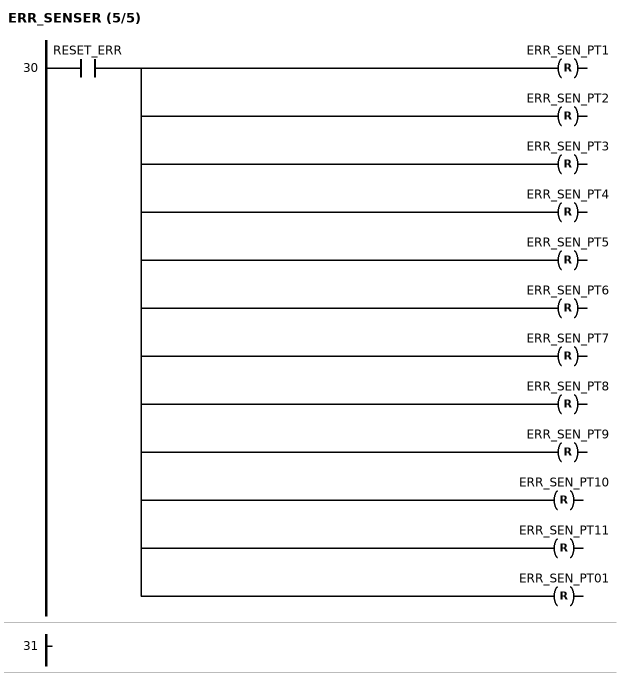
// NETWORK 30
ERR_SEN_PT1 R= RESET_ERR;
ERR_SEN_PT2 R= RESET_ERR;
ERR_SEN_PT3 R= RESET_ERR;
ERR_SEN_PT4 R= RESET_ERR;
ERR_SEN_PT5 R= RESET_ERR;
ERR_SEN_PT6 R= RESET_ERR;
ERR_SEN_PT7 R= RESET_ERR;
ERR_SEN_PT8 R= RESET_ERR;
ERR_SEN_PT9 R= RESET_ERR;
ERR_SEN_PT10 R= RESET_ERR;
ERR_SEN_PT11 R= RESET_ERR;
ERR_SEN_PT01 R= RESET_ERR;

// NETWORK 31

END_PROGRAM

// MyController/Application/SECURITY_BOILER
PROGRAM SECURITY_BOILER
VAR
END_VAR
VAR // added by the converter: edge detectors and wires of the graphical bodies
    _rt1, _rt2, _rt3, _rt4, _rt5 : R_TRIG;
END_VAR

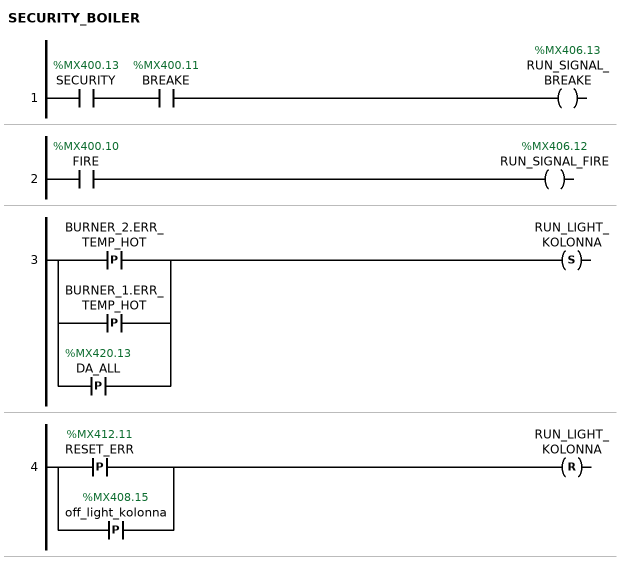
// NETWORK 1
//   SECURITY: AT %MX400.13
//   BREAKE: AT %MX400.11
//   RUN_SIGNAL_BREAKE: AT %MX406.13
RUN_SIGNAL_BREAKE := SECURITY AND BREAKE;

// NETWORK 2
//   FIRE: AT %MX400.10
//   RUN_SIGNAL_FIRE: AT %MX406.12
RUN_SIGNAL_FIRE := FIRE;

// NETWORK 3
//   DA_ALL: AT %MX420.13
_rt1(CLK := BURNER_2.ERR_TEMP_HOT);
_rt2(CLK := BURNER_1.ERR_TEMP_HOT);
_rt3(CLK := DA_ALL);
RUN_LIGHT_KOLONNA S= _rt1.Q OR _rt2.Q OR _rt3.Q;

// NETWORK 4
//   RESET_ERR: AT %MX412.11
//   off_light_kolonna: AT %MX408.15
_rt4(CLK := RESET_ERR);
_rt5(CLK := off_light_kolonna);
RUN_LIGHT_KOLONNA R= _rt4.Q OR _rt5.Q;

END_PROGRAM

// MyController/Application/VALVE_FEEDER_PUMP_FEEDERS_M3_M4
PROGRAM VALVE_FEEDER_PUMP_FEEDERS_M3_M4
VAR
	FEEDER_M3_CYCLE: BOOL;
	FEEDER_M4_CYCLE: BOOL;
	SMALL_PRESS: BOOL;
	run_feeder_to_open: BOOL;
END_VAR
VAR // added by the converter: edge detectors and wires of the graphical bodies
    _rt1, _rt2 : R_TRIG;
    _w1, _w2 : BOOL;
END_VAR

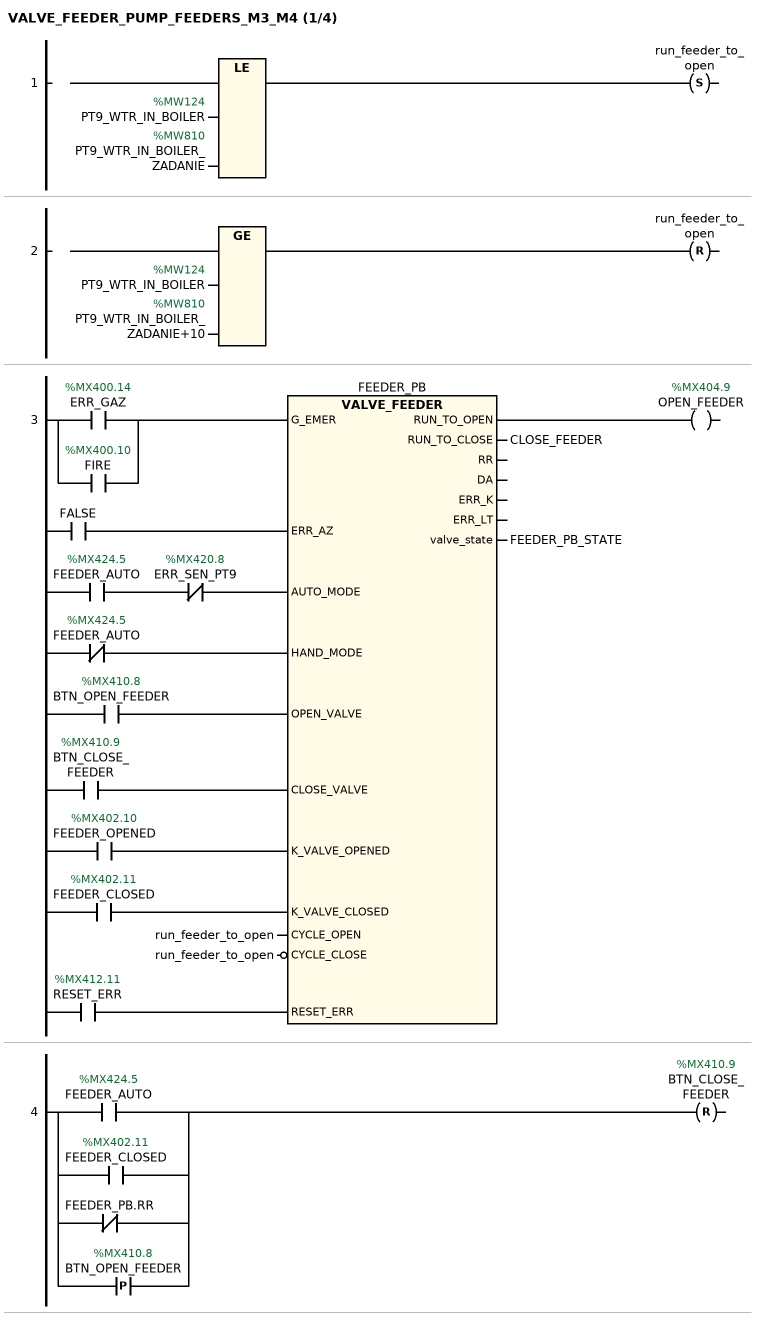
// NETWORK 1
//   PT9_WTR_IN_BOILER: AT %MW124
//   PT9_WTR_IN_BOILER_ZADANIE: AT %MW810
run_feeder_to_open S= PT9_WTR_IN_BOILER <= PT9_WTR_IN_BOILER_ZADANIE;

// NETWORK 2
//   PT9_WTR_IN_BOILER: AT %MW124
//   PT9_WTR_IN_BOILER_ZADANIE+10: AT %MW810
run_feeder_to_open R= PT9_WTR_IN_BOILER >= (PT9_WTR_IN_BOILER_ZADANIE+10);

// NETWORK 3
//   ERR_GAZ: AT %MX400.14
//   FIRE: AT %MX400.10
//   FEEDER_AUTO: AT %MX424.5
//   ERR_SEN_PT9: AT %MX420.8
//   BTN_OPEN_FEEDER: AT %MX410.8
//   BTN_CLOSE_FEEDER: AT %MX410.9
//   FEEDER_OPENED: AT %MX402.10
//   FEEDER_CLOSED: AT %MX402.11
//   RESET_ERR: AT %MX412.11
//   CLOSE_FEEDER: AT %MX404.10
//   FEEDER_PB_STATE: AT %MW406
//   OPEN_FEEDER: AT %MX404.9
FEEDER_PB(
    G_EMER := ERR_GAZ OR FIRE,
    ERR_AZ := FALSE,
    AUTO_MODE := FEEDER_AUTO AND NOT ERR_SEN_PT9,
    HAND_MODE := NOT FEEDER_AUTO,
    OPEN_VALVE := BTN_OPEN_FEEDER,
    CLOSE_VALVE := BTN_CLOSE_FEEDER,
    K_VALVE_OPENED := FEEDER_OPENED,
    K_VALVE_CLOSED := FEEDER_CLOSED,
    CYCLE_OPEN := run_feeder_to_open,
    CYCLE_CLOSE := NOT run_feeder_to_open,
    RESET_ERR := RESET_ERR,
    RUN_TO_CLOSE => CLOSE_FEEDER,
    valve_state => FEEDER_PB_STATE); // VALVE_FEEDER
OPEN_FEEDER := FEEDER_PB.RUN_TO_OPEN;

// NETWORK 4
//   FEEDER_AUTO: AT %MX424.5
//   FEEDER_CLOSED: AT %MX402.11
//   BTN_OPEN_FEEDER: AT %MX410.8
//   BTN_CLOSE_FEEDER: AT %MX410.9
_rt1(CLK := BTN_OPEN_FEEDER);
BTN_CLOSE_FEEDER R= FEEDER_AUTO OR FEEDER_CLOSED OR NOT FEEDER_PB.RR OR _rt1.Q;

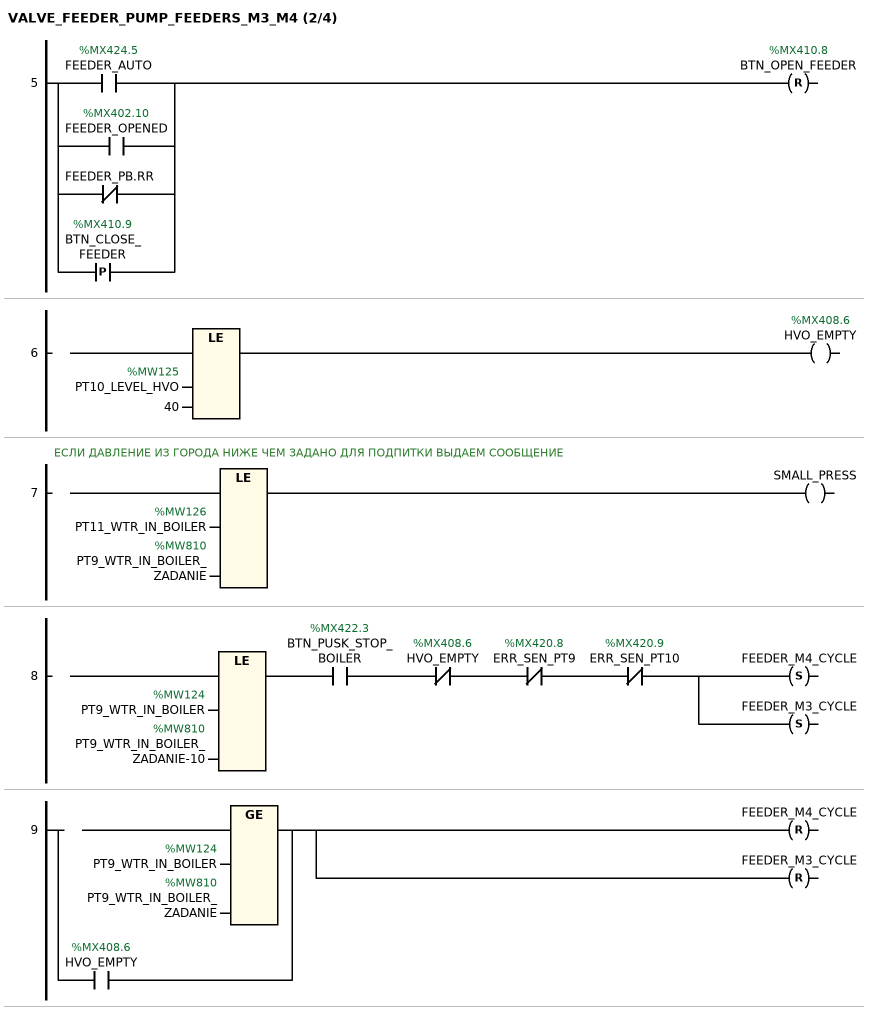
// NETWORK 5
//   FEEDER_AUTO: AT %MX424.5
//   FEEDER_OPENED: AT %MX402.10
//   BTN_CLOSE_FEEDER: AT %MX410.9
//   BTN_OPEN_FEEDER: AT %MX410.8
_rt2(CLK := BTN_CLOSE_FEEDER);
BTN_OPEN_FEEDER R= FEEDER_AUTO OR FEEDER_OPENED OR NOT FEEDER_PB.RR OR _rt2.Q;

// NETWORK 6
//   PT10_LEVEL_HVO: AT %MW125
//   HVO_EMPTY: AT %MX408.6
HVO_EMPTY := PT10_LEVEL_HVO <= 40;

// NETWORK 7
// ЕСЛИ ДАВЛЕНИЕ ИЗ ГОРОДА НИЖЕ ЧЕМ ЗАДАНО ДЛЯ ПОДПИТКИ ВЫДАЕМ СООБЩЕНИЕ
//   PT11_WTR_IN_BOILER: AT %MW126
//   PT9_WTR_IN_BOILER_ZADANIE: AT %MW810
SMALL_PRESS := PT11_WTR_IN_BOILER <= PT9_WTR_IN_BOILER_ZADANIE;

// NETWORK 8
//   PT9_WTR_IN_BOILER: AT %MW124
//   PT9_WTR_IN_BOILER_ZADANIE-10: AT %MW810
//   BTN_PUSK_STOP_BOILER: AT %MX422.3
//   HVO_EMPTY: AT %MX408.6
//   ERR_SEN_PT9: AT %MX420.8
//   ERR_SEN_PT10: AT %MX420.9
_w1 := PT9_WTR_IN_BOILER <= (PT9_WTR_IN_BOILER_ZADANIE-10) AND BTN_PUSK_STOP_BOILER AND NOT HVO_EMPTY AND NOT ERR_SEN_PT9 AND NOT ERR_SEN_PT10;
FEEDER_M4_CYCLE S= _w1;
FEEDER_M3_CYCLE S= _w1;

// NETWORK 9
//   PT9_WTR_IN_BOILER: AT %MW124
//   PT9_WTR_IN_BOILER_ZADANIE: AT %MW810
//   HVO_EMPTY: AT %MX408.6
_w2 := PT9_WTR_IN_BOILER >= PT9_WTR_IN_BOILER_ZADANIE OR HVO_EMPTY;
FEEDER_M4_CYCLE R= _w2;
FEEDER_M3_CYCLE R= _w2;

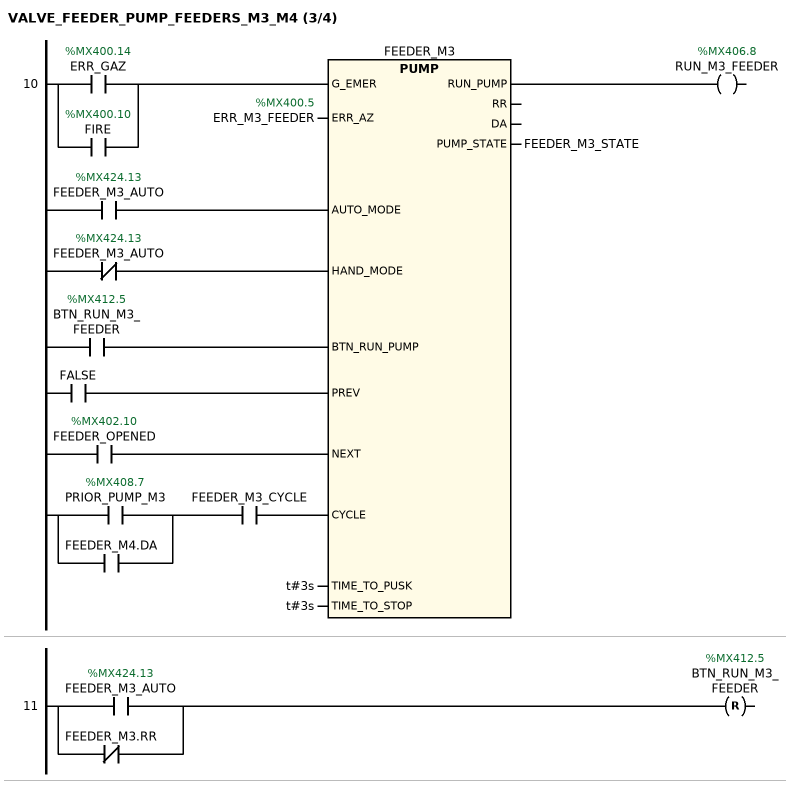
// NETWORK 10
//   ERR_GAZ: AT %MX400.14
//   FIRE: AT %MX400.10
//   ERR_M3_FEEDER: AT %MX400.5
//   FEEDER_M3_AUTO: AT %MX424.13
//   BTN_RUN_M3_FEEDER: AT %MX412.5
//   FEEDER_OPENED: AT %MX402.10
//   PRIOR_PUMP_M3: AT %MX408.7
//   FEEDER_M3_STATE: AT %MW411
//   RUN_M3_FEEDER: AT %MX406.8
FEEDER_M3(
    G_EMER := ERR_GAZ OR FIRE,
    ERR_AZ := ERR_M3_FEEDER,
    AUTO_MODE := FEEDER_M3_AUTO,
    HAND_MODE := NOT FEEDER_M3_AUTO,
    BTN_RUN_PUMP := BTN_RUN_M3_FEEDER,
    PREV := FALSE,
    NEXT := FEEDER_OPENED,
    CYCLE := (PRIOR_PUMP_M3 OR FEEDER_M4.DA) AND FEEDER_M3_CYCLE,
    TIME_TO_PUSK := t#3s,
    TIME_TO_STOP := t#3s,
    PUMP_STATE => FEEDER_M3_STATE); // PUMP
RUN_M3_FEEDER := FEEDER_M3.RUN_PUMP;

// NETWORK 11
//   FEEDER_M3_AUTO: AT %MX424.13
//   BTN_RUN_M3_FEEDER: AT %MX412.5
BTN_RUN_M3_FEEDER R= FEEDER_M3_AUTO OR NOT FEEDER_M3.RR;

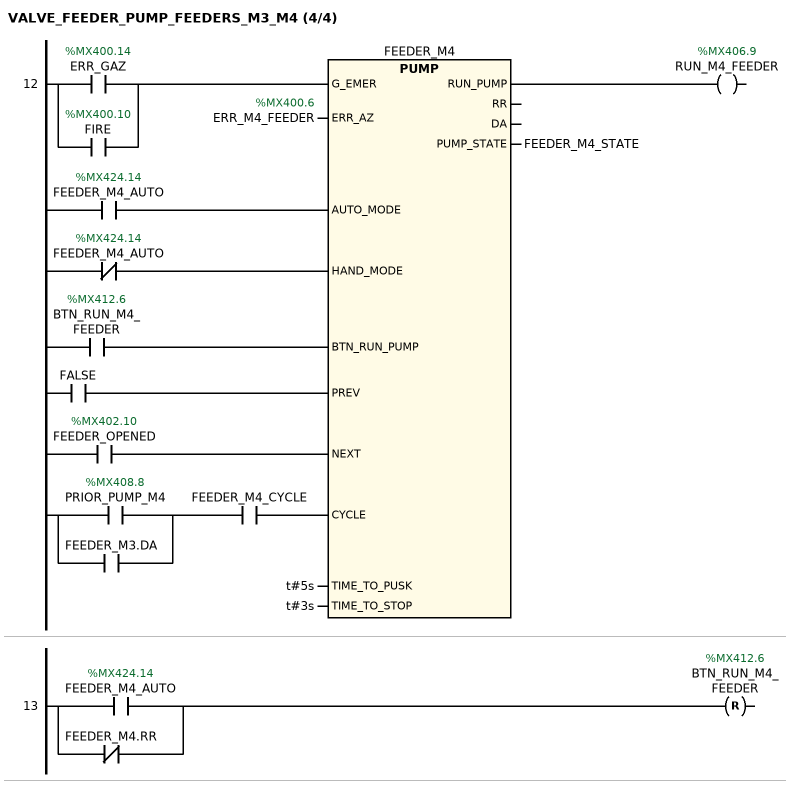
// NETWORK 12
//   ERR_GAZ: AT %MX400.14
//   FIRE: AT %MX400.10
//   ERR_M4_FEEDER: AT %MX400.6
//   FEEDER_M4_AUTO: AT %MX424.14
//   BTN_RUN_M4_FEEDER: AT %MX412.6
//   FEEDER_OPENED: AT %MX402.10
//   PRIOR_PUMP_M4: AT %MX408.8
//   FEEDER_M4_STATE: AT %MW412
//   RUN_M4_FEEDER: AT %MX406.9
FEEDER_M4(
    G_EMER := ERR_GAZ OR FIRE,
    ERR_AZ := ERR_M4_FEEDER,
    AUTO_MODE := FEEDER_M4_AUTO,
    HAND_MODE := NOT FEEDER_M4_AUTO,
    BTN_RUN_PUMP := BTN_RUN_M4_FEEDER,
    PREV := FALSE,
    NEXT := FEEDER_OPENED,
    CYCLE := (PRIOR_PUMP_M4 OR FEEDER_M3.DA) AND FEEDER_M4_CYCLE,
    TIME_TO_PUSK := t#5s,
    TIME_TO_STOP := t#3s,
    PUMP_STATE => FEEDER_M4_STATE); // PUMP
RUN_M4_FEEDER := FEEDER_M4.RUN_PUMP;

// NETWORK 13
//   FEEDER_M4_AUTO: AT %MX424.14
//   BTN_RUN_M4_FEEDER: AT %MX412.6
BTN_RUN_M4_FEEDER R= FEEDER_M4_AUTO OR NOT FEEDER_M4.RR;

END_PROGRAM

// MyController/Application/FB/VALVE_FEEDER
FUNCTION_BLOCK VALVE_FEEDER
VAR_INPUT
	G_EMER: BOOL;
	ERR_AZ: BOOL;
	AUTO_MODE: BOOL;
	HAND_MODE: BOOL;
	OPEN_VALVE: BOOL;
	CLOSE_VALVE: BOOL;
	K_VALVE_OPENED: BOOL;
	K_VALVE_CLOSED: BOOL;
	CYCLE_OPEN: BOOL;
	CYCLE_CLOSE: BOOL;
	RESET_ERR: BOOL;	
END_VAR
VAR_OUTPUT
	RUN_TO_OPEN: BOOL;
	RUN_TO_CLOSE: BOOL;
	RR: BOOL;
	DA: BOOL;
	ERR_K: BOOL;
	ERR_LT: BOOL;
	valve_state: BYTE;
END_VAR
VAR
	TM_LT_VALVE: TON;
	tm_err_k: TOF;
END_VAR
VAR // added by the converter: edge detectors and wires of the graphical bodies
    _w1 : BOOL;
END_VAR

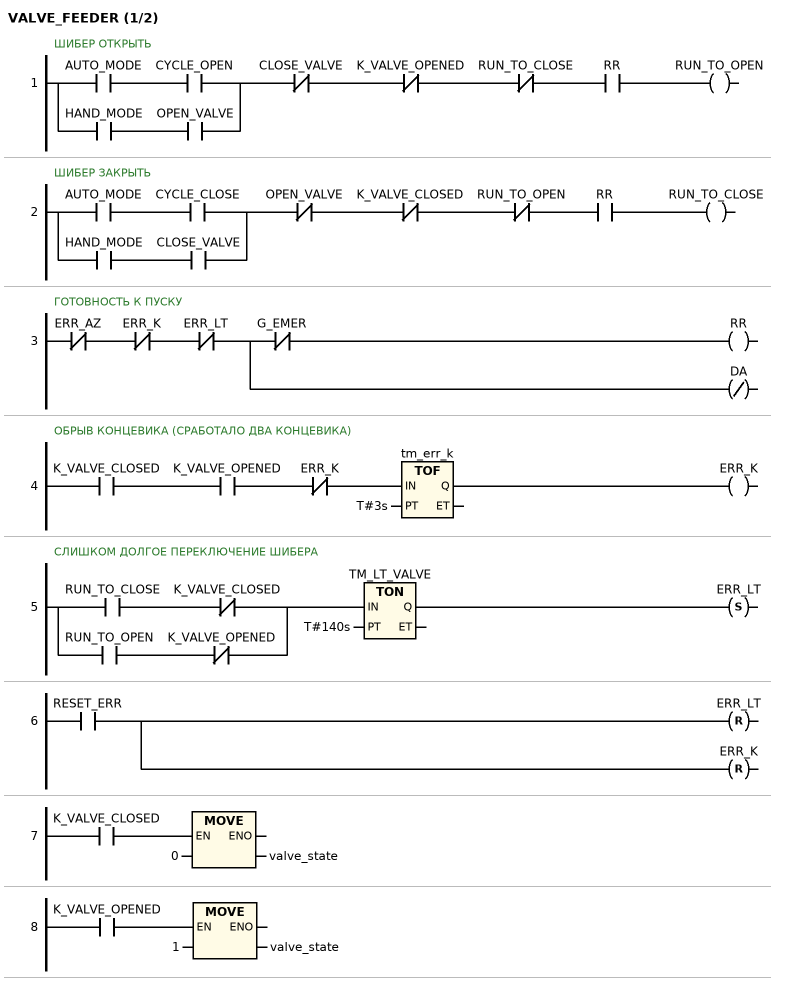
// NETWORK 1
// ШИБЕР ОТКРЫТЬ
RUN_TO_OPEN := (AUTO_MODE AND CYCLE_OPEN OR HAND_MODE AND OPEN_VALVE) AND NOT CLOSE_VALVE AND NOT K_VALVE_OPENED AND NOT RUN_TO_CLOSE AND RR;

// NETWORK 2
// ШИБЕР ЗАКРЫТЬ
RUN_TO_CLOSE := (AUTO_MODE AND CYCLE_CLOSE OR HAND_MODE AND CLOSE_VALVE) AND NOT OPEN_VALVE AND NOT K_VALVE_CLOSED AND NOT RUN_TO_OPEN AND RR;

// NETWORK 3
// ГОТОВНОСТЬ К ПУСКУ
_w1 := NOT ERR_AZ AND NOT ERR_K AND NOT ERR_LT;
RR := _w1 AND NOT G_EMER;
DA := NOT _w1;

// NETWORK 4
// ОБРЫВ КОНЦЕВИКА (СРАБОТАЛО ДВА КОНЦЕВИКА)
tm_err_k(IN := K_VALVE_CLOSED AND K_VALVE_OPENED AND NOT ERR_K, PT := T#3s); // TOF
ERR_K := tm_err_k.Q;

// NETWORK 5
// СЛИШКОМ ДОЛГОЕ ПЕРЕКЛЮЧЕНИЕ ШИБЕРА
TM_LT_VALVE(IN := RUN_TO_CLOSE AND NOT K_VALVE_CLOSED OR RUN_TO_OPEN AND NOT K_VALVE_OPENED, PT := T#140s); // TON
ERR_LT S= TM_LT_VALVE.Q;

// NETWORK 6
ERR_LT R= RESET_ERR;
ERR_K R= RESET_ERR;

// NETWORK 7
IF K_VALVE_CLOSED THEN valve_state := 0; END_IF

// NETWORK 8
IF K_VALVE_OPENED THEN valve_state := 1; END_IF

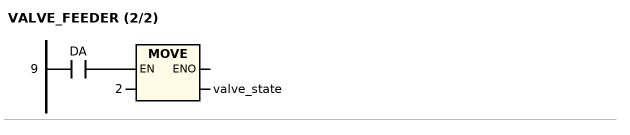
// NETWORK 9
IF DA THEN valve_state := 2; END_IF

END_FUNCTION_BLOCK

// MyController/Application/NET_PUMPS_M1_M2
PROGRAM NET_PUMPS_M1_M2
VAR
	PUMP_M1_CYCLE: BOOL;
	PUMP_M2_CYCLE: BOOL;
	TM_ERR_FLOW_WATER_IN_NET: TON;
	
	TON_0: TON;
	PID_M1: PID;
	PID_M2: PID;
END_VAR

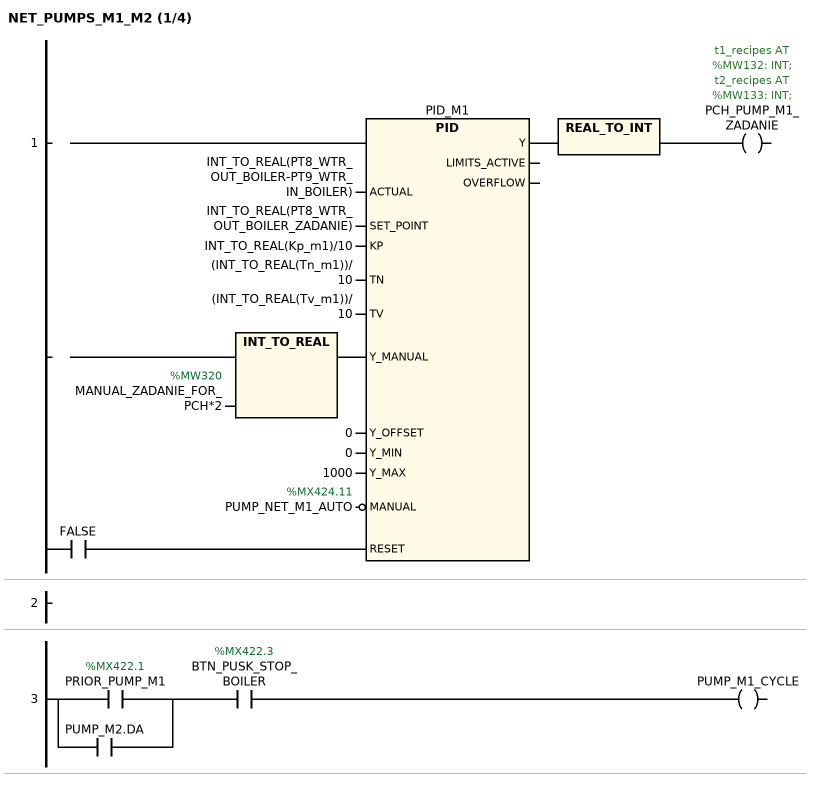
// NETWORK 1
//   MANUAL_ZADANIE_FOR_PCH*2: Задание для М1 | AT %MW320
//   PUMP_NET_M1_AUTO: AT %MX424.11
//   PCH_PUMP_M1_ZADANIE: t1_recipes AT %MW132: INT; t2_recipes AT %MW133: INT;
PID_M1(
    ACTUAL := INT_TO_REAL(PT8_WTR_OUT_BOILER-PT9_WTR_IN_BOILER),
    SET_POINT := INT_TO_REAL(PT8_WTR_OUT_BOILER_ZADANIE),
    KP := INT_TO_REAL(Kp_m1)/10,
    TN := (INT_TO_REAL(Tn_m1))/10,
    TV := (INT_TO_REAL(Tv_m1))/10,
    Y_MANUAL := INT_TO_REAL(MANUAL_ZADANIE_FOR_PCH*2),
    Y_OFFSET := 0,
    Y_MIN := 0,
    Y_MAX := 1000,
    MANUAL := NOT PUMP_NET_M1_AUTO,
    RESET := FALSE); // PID
PCH_PUMP_M1_ZADANIE := REAL_TO_INT(PID_M1.Y);

// NETWORK 2

// NETWORK 3
//   PRIOR_PUMP_M1: AT %MX422.1
//   BTN_PUSK_STOP_BOILER: AT %MX422.3
PUMP_M1_CYCLE := (PRIOR_PUMP_M1 OR PUMP_M2.DA) AND BTN_PUSK_STOP_BOILER;

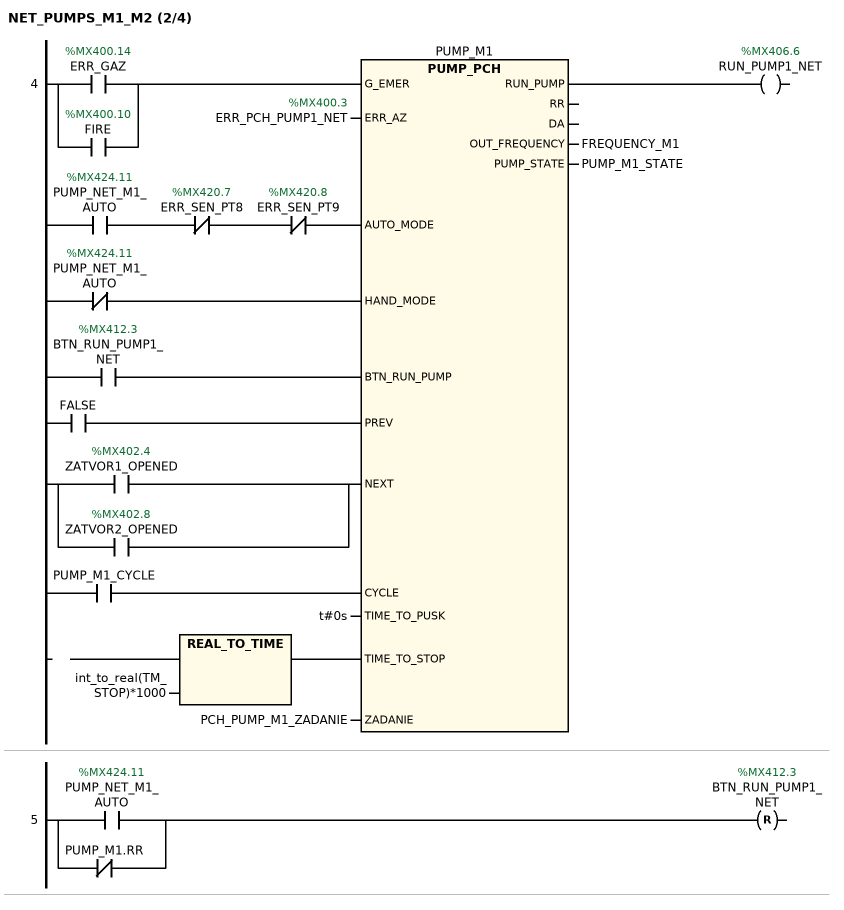
// NETWORK 4
//   ERR_GAZ: AT %MX400.14
//   FIRE: AT %MX400.10
//   ERR_PCH_PUMP1_NET: AT %MX400.3
//   PUMP_NET_M1_AUTO: AT %MX424.11
//   ERR_SEN_PT8: AT %MX420.7
//   ERR_SEN_PT9: AT %MX420.8
//   BTN_RUN_PUMP1_NET: AT %MX412.3
//   ZATVOR1_OPENED: AT %MX402.4
//   ZATVOR2_OPENED: AT %MX402.8
//   PCH_PUMP_M1_ZADANIE: t1_recipes AT %MW132: INT; t2_recipes AT %MW133: INT;
//   FREQUENCY_M1: AT %MW134
//   PUMP_M1_STATE: AT %MW409
//   RUN_PUMP1_NET: AT %MX406.6
PUMP_M1(
    G_EMER := ERR_GAZ OR FIRE,
    ERR_AZ := ERR_PCH_PUMP1_NET,
    AUTO_MODE := PUMP_NET_M1_AUTO AND NOT ERR_SEN_PT8 AND NOT ERR_SEN_PT9,
    HAND_MODE := NOT PUMP_NET_M1_AUTO,
    BTN_RUN_PUMP := BTN_RUN_PUMP1_NET,
    PREV := FALSE,
    NEXT := ZATVOR1_OPENED OR ZATVOR2_OPENED,
    CYCLE := PUMP_M1_CYCLE,
    TIME_TO_PUSK := t#0s,
    TIME_TO_STOP := REAL_TO_TIME(int_to_real(TM_STOP)*1000),
    ZADANIE := PCH_PUMP_M1_ZADANIE,
    OUT_FREQUENCY => FREQUENCY_M1,
    PUMP_STATE => PUMP_M1_STATE); // PUMP_PCH
RUN_PUMP1_NET := PUMP_M1.RUN_PUMP;

// NETWORK 5
//   PUMP_NET_M1_AUTO: AT %MX424.11
//   BTN_RUN_PUMP1_NET: AT %MX412.3
BTN_RUN_PUMP1_NET R= PUMP_NET_M1_AUTO OR NOT PUMP_M1.RR;

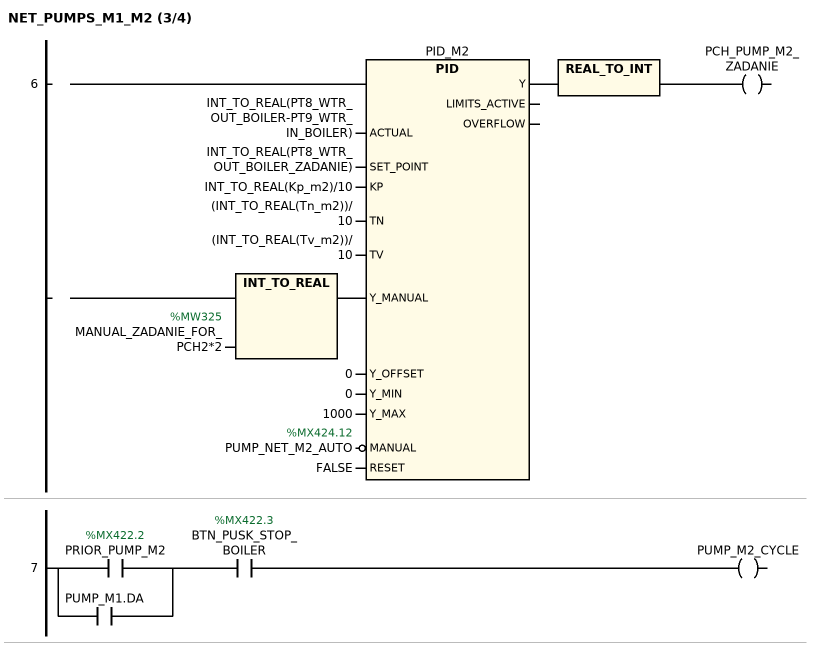
// NETWORK 6
//   MANUAL_ZADANIE_FOR_PCH2*2: Задание для М2 | AT %MW325
//   PUMP_NET_M2_AUTO: AT %MX424.12
PID_M2(
    ACTUAL := INT_TO_REAL(PT8_WTR_OUT_BOILER-PT9_WTR_IN_BOILER),
    SET_POINT := INT_TO_REAL(PT8_WTR_OUT_BOILER_ZADANIE),
    KP := INT_TO_REAL(Kp_m2)/10,
    TN := (INT_TO_REAL(Tn_m2))/10,
    TV := (INT_TO_REAL(Tv_m2))/10,
    Y_MANUAL := INT_TO_REAL(MANUAL_ZADANIE_FOR_PCH2*2),
    Y_OFFSET := 0,
    Y_MIN := 0,
    Y_MAX := 1000,
    MANUAL := NOT PUMP_NET_M2_AUTO,
    RESET := FALSE); // PID
PCH_PUMP_M2_ZADANIE := REAL_TO_INT(PID_M2.Y);

// NETWORK 7
//   PRIOR_PUMP_M2: AT %MX422.2
//   BTN_PUSK_STOP_BOILER: AT %MX422.3
PUMP_M2_CYCLE := (PRIOR_PUMP_M2 OR PUMP_M1.DA) AND BTN_PUSK_STOP_BOILER;

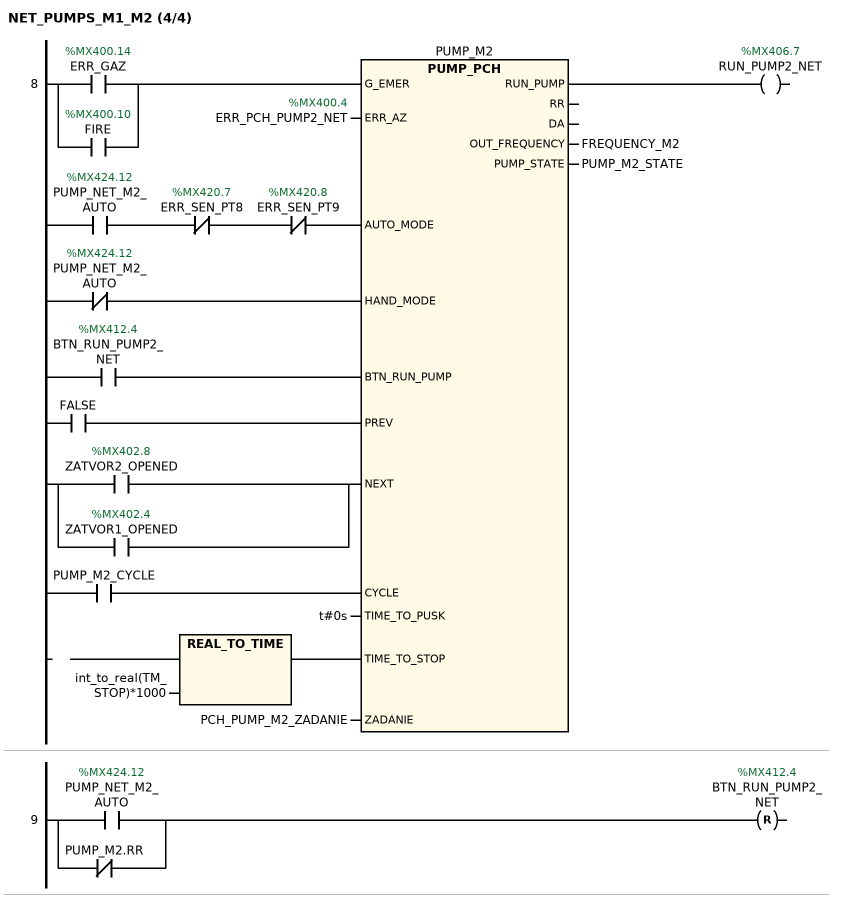
// NETWORK 8
//   ERR_GAZ: AT %MX400.14
//   FIRE: AT %MX400.10
//   ERR_PCH_PUMP2_NET: AT %MX400.4
//   PUMP_NET_M2_AUTO: AT %MX424.12
//   ERR_SEN_PT8: AT %MX420.7
//   ERR_SEN_PT9: AT %MX420.8
//   BTN_RUN_PUMP2_NET: AT %MX412.4
//   ZATVOR2_OPENED: AT %MX402.8
//   ZATVOR1_OPENED: AT %MX402.4
//   FREQUENCY_M2: AT %MW135
//   PUMP_M2_STATE: AT %MW410
//   RUN_PUMP2_NET: AT %MX406.7
PUMP_M2(
    G_EMER := ERR_GAZ OR FIRE,
    ERR_AZ := ERR_PCH_PUMP2_NET,
    AUTO_MODE := PUMP_NET_M2_AUTO AND NOT ERR_SEN_PT8 AND NOT ERR_SEN_PT9,
    HAND_MODE := NOT PUMP_NET_M2_AUTO,
    BTN_RUN_PUMP := BTN_RUN_PUMP2_NET,
    PREV := FALSE,
    NEXT := ZATVOR2_OPENED OR ZATVOR1_OPENED,
    CYCLE := PUMP_M2_CYCLE,
    TIME_TO_PUSK := t#0s,
    TIME_TO_STOP := REAL_TO_TIME(int_to_real(TM_STOP)*1000),
    ZADANIE := PCH_PUMP_M2_ZADANIE,
    OUT_FREQUENCY => FREQUENCY_M2,
    PUMP_STATE => PUMP_M2_STATE); // PUMP_PCH
RUN_PUMP2_NET := PUMP_M2.RUN_PUMP;

// NETWORK 9
//   PUMP_NET_M2_AUTO: AT %MX424.12
//   BTN_RUN_PUMP2_NET: AT %MX412.4
BTN_RUN_PUMP2_NET R= PUMP_NET_M2_AUTO OR NOT PUMP_M2.RR;

END_PROGRAM

// MyController/Application/TRHD_PEREPUSK
PROGRAM TRHD_PEREPUSK
VAR
	PID_PEREPUSK: PID;
	BLINK_FOR_PEREPUSK: BLINK;
	sTT: LIN_TRAFO;
END_VAR

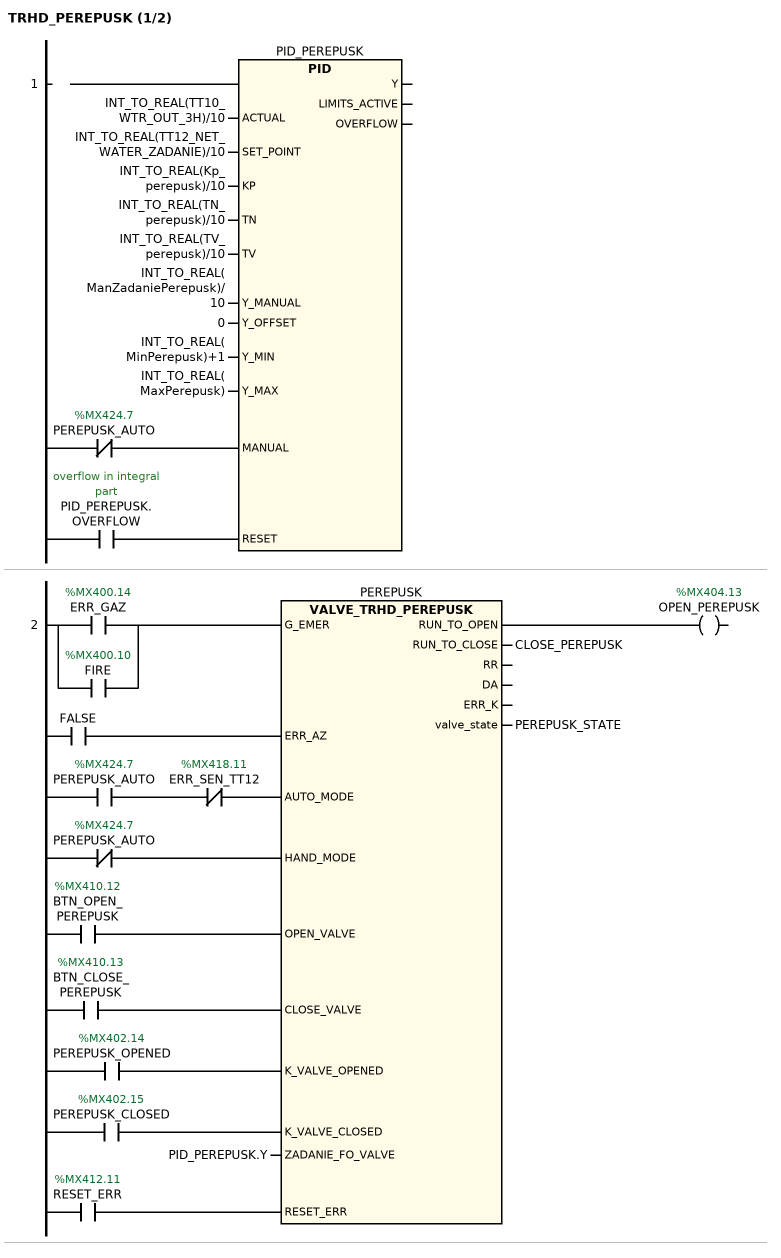
// NETWORK 1
//   PEREPUSK_AUTO: AT %MX424.7
//   PID_PEREPUSK.OVERFLOW: overflow in integral part
PID_PEREPUSK(
    ACTUAL := INT_TO_REAL(TT10_WTR_OUT_3H)/10,
    SET_POINT := INT_TO_REAL(TT12_NET_WATER_ZADANIE)/10,
    KP := INT_TO_REAL(Kp_perepusk)/10,
    TN := INT_TO_REAL(TN_perepusk)/10,
    TV := INT_TO_REAL(TV_perepusk)/10,
    Y_MANUAL := INT_TO_REAL(ManZadaniePerepusk)/10,
    Y_OFFSET := 0,
    Y_MIN := INT_TO_REAL(MinPerepusk)+1,
    Y_MAX := INT_TO_REAL(MaxPerepusk),
    MANUAL := NOT PEREPUSK_AUTO,
    RESET := PID_PEREPUSK.OVERFLOW); // PID

// NETWORK 2
//   ERR_GAZ: AT %MX400.14
//   FIRE: AT %MX400.10
//   PEREPUSK_AUTO: AT %MX424.7
//   ERR_SEN_TT12: AT %MX418.11
//   BTN_OPEN_PEREPUSK: AT %MX410.12
//   BTN_CLOSE_PEREPUSK: AT %MX410.13
//   PEREPUSK_OPENED: AT %MX402.14
//   PEREPUSK_CLOSED: AT %MX402.15
//   PID_PEREPUSK.Y: manipulated variable, set value
//   RESET_ERR: AT %MX412.11
//   CLOSE_PEREPUSK: AT %MX404.14
//   PEREPUSK_STATE: AT %MW405
//   OPEN_PEREPUSK: AT %MX404.13
PEREPUSK(
    G_EMER := ERR_GAZ OR FIRE,
    ERR_AZ := FALSE,
    AUTO_MODE := PEREPUSK_AUTO AND NOT ERR_SEN_TT12,
    HAND_MODE := NOT PEREPUSK_AUTO,
    OPEN_VALVE := BTN_OPEN_PEREPUSK,
    CLOSE_VALVE := BTN_CLOSE_PEREPUSK,
    K_VALVE_OPENED := PEREPUSK_OPENED,
    K_VALVE_CLOSED := PEREPUSK_CLOSED,
    ZADANIE_FO_VALVE := PID_PEREPUSK.Y,
    RESET_ERR := RESET_ERR,
    RUN_TO_CLOSE => CLOSE_PEREPUSK,
    valve_state => PEREPUSK_STATE); // VALVE_TRHD_PEREPUSK
OPEN_PEREPUSK := PEREPUSK.RUN_TO_OPEN;

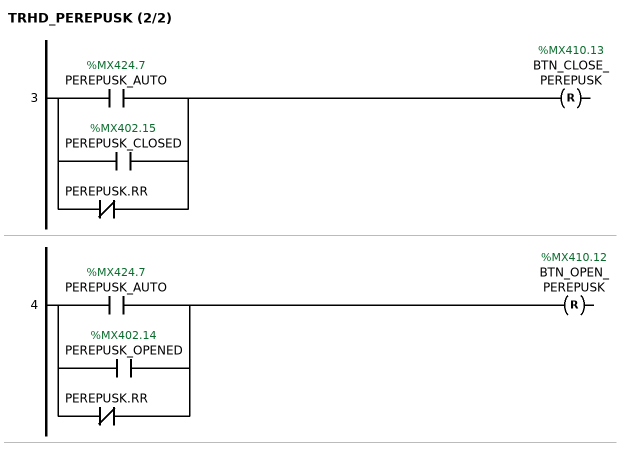
// NETWORK 3
//   PEREPUSK_AUTO: AT %MX424.7
//   PEREPUSK_CLOSED: AT %MX402.15
//   BTN_CLOSE_PEREPUSK: AT %MX410.13
BTN_CLOSE_PEREPUSK R= PEREPUSK_AUTO OR PEREPUSK_CLOSED OR NOT PEREPUSK.RR;

// NETWORK 4
//   PEREPUSK_AUTO: AT %MX424.7
//   PEREPUSK_OPENED: AT %MX402.14
//   BTN_OPEN_PEREPUSK: AT %MX410.12
BTN_OPEN_PEREPUSK R= PEREPUSK_AUTO OR PEREPUSK_OPENED OR NOT PEREPUSK.RR;

END_PROGRAM

// MyController/Application/FB/VALVE_TRHD_PEREPUSK
FUNCTION_BLOCK VALVE_TRHD_PEREPUSK
VAR_INPUT
	G_EMER: BOOL;
	ERR_AZ: BOOL;
	AUTO_MODE: BOOL;
	HAND_MODE: BOOL;
	OPEN_VALVE: BOOL;
	CLOSE_VALVE: BOOL;
	K_VALVE_OPENED: BOOL;
	K_VALVE_CLOSED: BOOL;
	ZADANIE_FO_VALVE: REAL;
	RESET_ERR: BOOL;	
END_VAR
VAR_OUTPUT
	RUN_TO_OPEN: BOOL;
	RUN_TO_CLOSE: BOOL;
	RR: BOOL;
	DA: BOOL;
	ERR_K: BOOL;
	valve_state: BYTE;
END_VAR
VAR
	TM_LT_VALVE: TON;
	RUN_VALVE_TO_OPEN: BOOL;
	CYCLE_OPEN: BOOL;
	CYCLE_CLOSE: BOOL;
END_VAR
VAR // added by the converter: edge detectors and wires of the graphical bodies
    _w1 : BOOL;
END_VAR

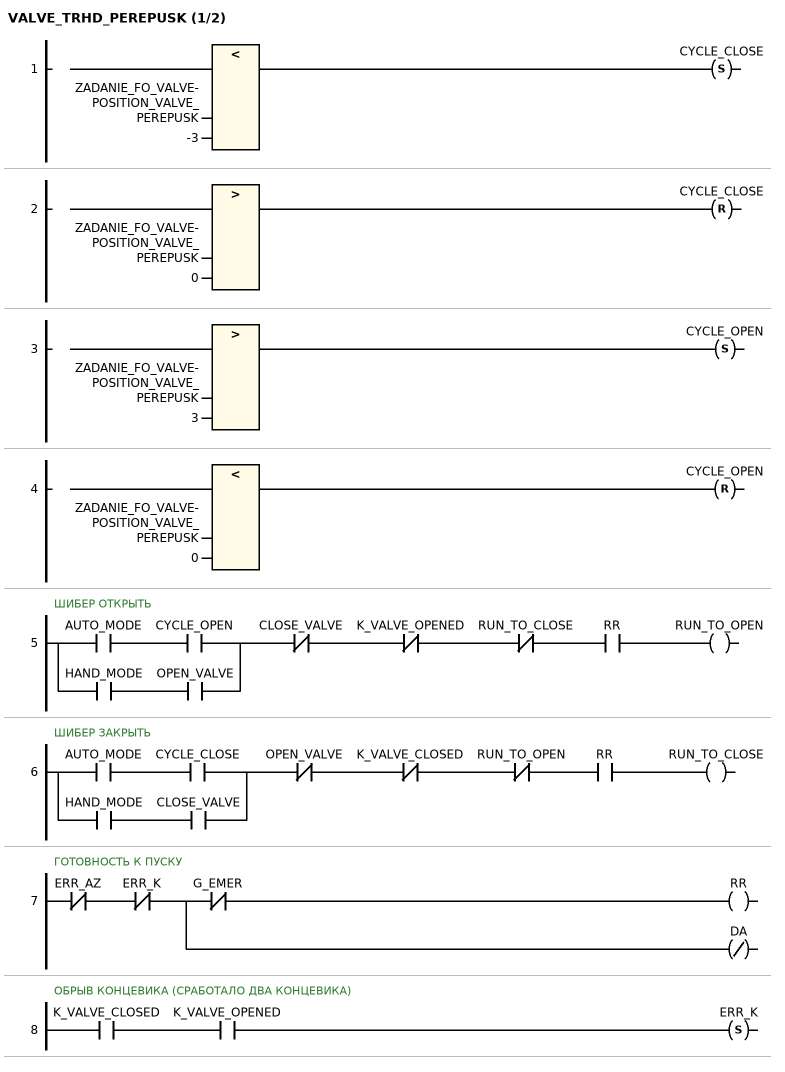
// NETWORK 1
CYCLE_CLOSE S= (ZADANIE_FO_VALVE-POSITION_VALVE_PEREPUSK) < -3;

// NETWORK 2
CYCLE_CLOSE R= (ZADANIE_FO_VALVE-POSITION_VALVE_PEREPUSK) > 0;

// NETWORK 3
CYCLE_OPEN S= (ZADANIE_FO_VALVE-POSITION_VALVE_PEREPUSK) > 3;

// NETWORK 4
CYCLE_OPEN R= (ZADANIE_FO_VALVE-POSITION_VALVE_PEREPUSK) < 0;

// NETWORK 5
// ШИБЕР ОТКРЫТЬ
RUN_TO_OPEN := (AUTO_MODE AND CYCLE_OPEN OR HAND_MODE AND OPEN_VALVE) AND NOT CLOSE_VALVE AND NOT K_VALVE_OPENED AND NOT RUN_TO_CLOSE AND RR;

// NETWORK 6
// ШИБЕР ЗАКРЫТЬ
RUN_TO_CLOSE := (AUTO_MODE AND CYCLE_CLOSE OR HAND_MODE AND CLOSE_VALVE) AND NOT OPEN_VALVE AND NOT K_VALVE_CLOSED AND NOT RUN_TO_OPEN AND RR;

// NETWORK 7
// ГОТОВНОСТЬ К ПУСКУ
_w1 := NOT ERR_AZ AND NOT ERR_K;
RR := _w1 AND NOT G_EMER;
DA := NOT _w1;

// NETWORK 8
// ОБРЫВ КОНЦЕВИКА (СРАБОТАЛО ДВА КОНЦЕВИКА)
ERR_K S= K_VALVE_CLOSED AND K_VALVE_OPENED;

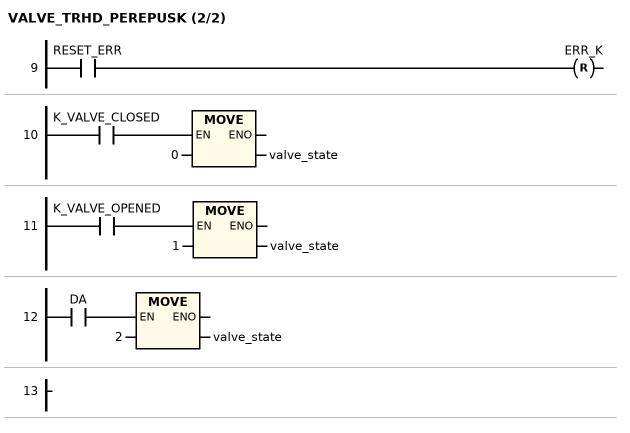
// NETWORK 9
ERR_K R= RESET_ERR;

// NETWORK 10
IF K_VALVE_CLOSED THEN valve_state := 0; END_IF

// NETWORK 11
IF K_VALVE_OPENED THEN valve_state := 1; END_IF

// NETWORK 12
IF DA THEN valve_state := 2; END_IF

// NETWORK 13

END_FUNCTION_BLOCK

// MyController/Application/ZATVORS
PROGRAM ZATVORS
VAR
	TM_CLOSE_ZATVOR_1: TOF;
	TM_CLOSE_ZATVOR_2: TOF;;
	
	
	ZATVOR_BURNER2_CYCLE_OPEN: BOOL;
	ZATVOR_BURNER2_CYCLE_CLOSE: BOOL;
	ZATVOR_BURNER1_CYCLE_OPEN: BOOL;
	ZATVOR_BURNER1_CYCLE_CLOSE: BOOL;
	
	tm_flow2: TON;
	tm_fl1: TON;
END_VAR
VAR // added by the converter: edge detectors and wires of the graphical bodies
    _rt1, _rt2, _rt3, _rt4 : R_TRIG;
END_VAR

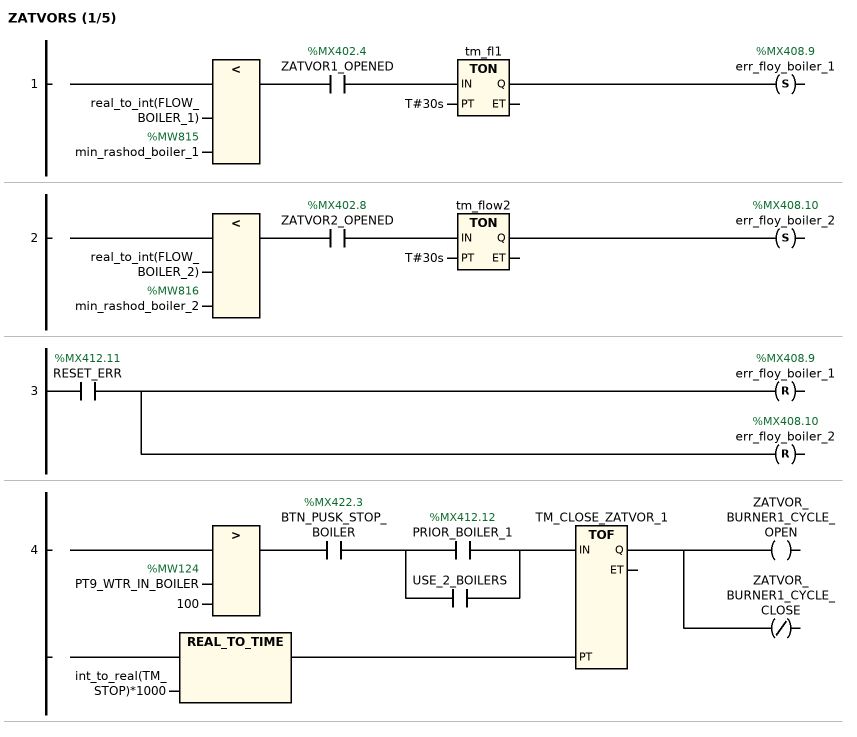
// NETWORK 1
//   min_rashod_boiler_1: AT %MW815
//   ZATVOR1_OPENED: AT %MX402.4
//   err_floy_boiler_1: AT %MX408.9
tm_fl1(IN := (real_to_int(FLOW_BOILER_1)) < min_rashod_boiler_1 AND ZATVOR1_OPENED, PT := T#30s); // TON
err_floy_boiler_1 S= tm_fl1.Q;

// NETWORK 2
//   min_rashod_boiler_2: AT %MW816
//   ZATVOR2_OPENED: AT %MX402.8
//   err_floy_boiler_2: AT %MX408.10
tm_flow2(IN := (real_to_int(FLOW_BOILER_2)) < min_rashod_boiler_2 AND ZATVOR2_OPENED, PT := T#30s); // TON
err_floy_boiler_2 S= tm_flow2.Q;

// NETWORK 3
//   RESET_ERR: AT %MX412.11
//   err_floy_boiler_1: AT %MX408.9
//   err_floy_boiler_2: AT %MX408.10
err_floy_boiler_1 R= RESET_ERR;
err_floy_boiler_2 R= RESET_ERR;

// NETWORK 4
//   PT9_WTR_IN_BOILER: AT %MW124
//   BTN_PUSK_STOP_BOILER: AT %MX422.3
//   PRIOR_BOILER_1: AT %MX412.12
TM_CLOSE_ZATVOR_1(IN := PT9_WTR_IN_BOILER > 100 AND BTN_PUSK_STOP_BOILER AND (PRIOR_BOILER_1 OR USE_2_BOILERS), PT := REAL_TO_TIME(int_to_real(TM_STOP)*1000)); // TOF
ZATVOR_BURNER1_CYCLE_OPEN := TM_CLOSE_ZATVOR_1.Q;
ZATVOR_BURNER1_CYCLE_CLOSE := NOT TM_CLOSE_ZATVOR_1.Q;

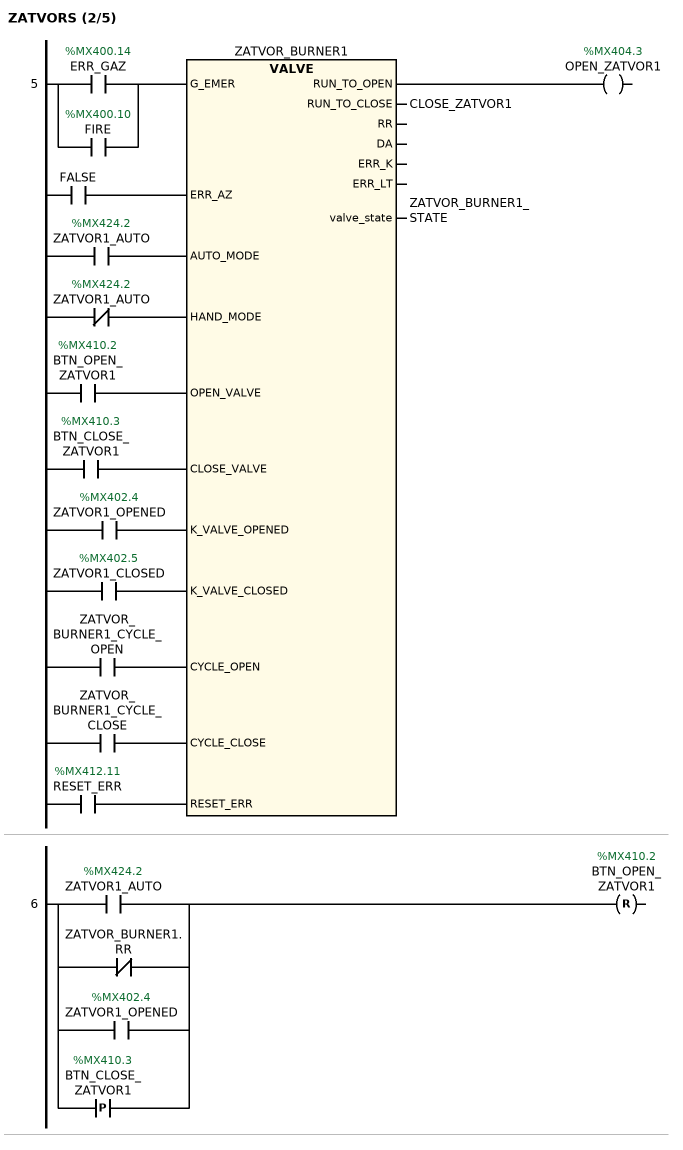
// NETWORK 5
//   ERR_GAZ: AT %MX400.14
//   FIRE: AT %MX400.10
//   ZATVOR1_AUTO: AT %MX424.2
//   BTN_OPEN_ZATVOR1: AT %MX410.2
//   BTN_CLOSE_ZATVOR1: AT %MX410.3
//   ZATVOR1_OPENED: AT %MX402.4
//   ZATVOR1_CLOSED: AT %MX402.5
//   RESET_ERR: AT %MX412.11
//   CLOSE_ZATVOR1: AT %MX404.4
//   ZATVOR_BURNER1_STATE: AT %MW407
//   OPEN_ZATVOR1: AT %MX404.3
ZATVOR_BURNER1(
    G_EMER := ERR_GAZ OR FIRE,
    ERR_AZ := FALSE,
    AUTO_MODE := ZATVOR1_AUTO,
    HAND_MODE := NOT ZATVOR1_AUTO,
    OPEN_VALVE := BTN_OPEN_ZATVOR1,
    CLOSE_VALVE := BTN_CLOSE_ZATVOR1,
    K_VALVE_OPENED := ZATVOR1_OPENED,
    K_VALVE_CLOSED := ZATVOR1_CLOSED,
    CYCLE_OPEN := ZATVOR_BURNER1_CYCLE_OPEN,
    CYCLE_CLOSE := ZATVOR_BURNER1_CYCLE_CLOSE,
    RESET_ERR := RESET_ERR,
    RUN_TO_CLOSE => CLOSE_ZATVOR1,
    valve_state => ZATVOR_BURNER1_STATE); // VALVE
OPEN_ZATVOR1 := ZATVOR_BURNER1.RUN_TO_OPEN;

// NETWORK 6
//   ZATVOR1_AUTO: AT %MX424.2
//   ZATVOR1_OPENED: AT %MX402.4
//   BTN_CLOSE_ZATVOR1: AT %MX410.3
//   BTN_OPEN_ZATVOR1: AT %MX410.2
_rt1(CLK := BTN_CLOSE_ZATVOR1);
BTN_OPEN_ZATVOR1 R= ZATVOR1_AUTO OR NOT ZATVOR_BURNER1.RR OR ZATVOR1_OPENED OR _rt1.Q;

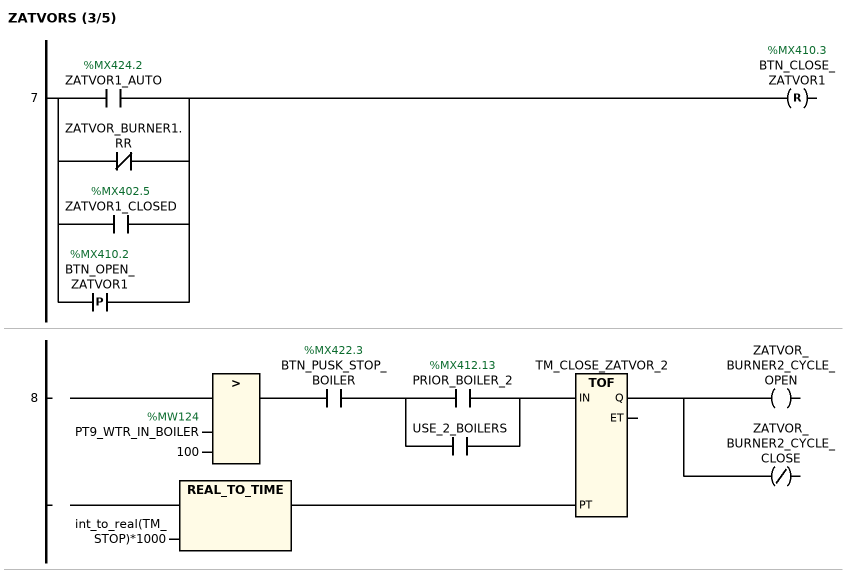
// NETWORK 7
//   ZATVOR1_AUTO: AT %MX424.2
//   ZATVOR1_CLOSED: AT %MX402.5
//   BTN_OPEN_ZATVOR1: AT %MX410.2
//   BTN_CLOSE_ZATVOR1: AT %MX410.3
_rt2(CLK := BTN_OPEN_ZATVOR1);
BTN_CLOSE_ZATVOR1 R= ZATVOR1_AUTO OR NOT ZATVOR_BURNER1.RR OR ZATVOR1_CLOSED OR _rt2.Q;

// NETWORK 8
//   PT9_WTR_IN_BOILER: AT %MW124
//   BTN_PUSK_STOP_BOILER: AT %MX422.3
//   PRIOR_BOILER_2: AT %MX412.13
TM_CLOSE_ZATVOR_2(IN := PT9_WTR_IN_BOILER > 100 AND BTN_PUSK_STOP_BOILER AND (PRIOR_BOILER_2 OR USE_2_BOILERS), PT := REAL_TO_TIME(int_to_real(TM_STOP)*1000)); // TOF
ZATVOR_BURNER2_CYCLE_OPEN := TM_CLOSE_ZATVOR_2.Q;
ZATVOR_BURNER2_CYCLE_CLOSE := NOT TM_CLOSE_ZATVOR_2.Q;

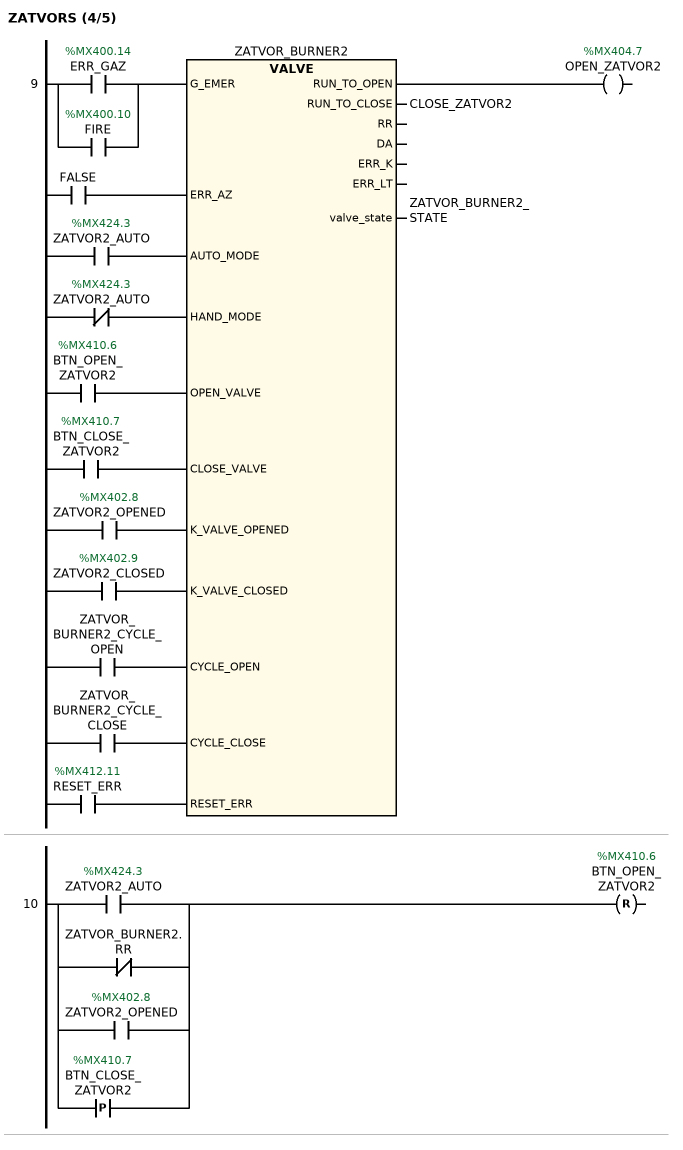
// NETWORK 9
//   ERR_GAZ: AT %MX400.14
//   FIRE: AT %MX400.10
//   ZATVOR2_AUTO: AT %MX424.3
//   BTN_OPEN_ZATVOR2: AT %MX410.6
//   BTN_CLOSE_ZATVOR2: AT %MX410.7
//   ZATVOR2_OPENED: AT %MX402.8
//   ZATVOR2_CLOSED: AT %MX402.9
//   RESET_ERR: AT %MX412.11
//   CLOSE_ZATVOR2: AT %MX404.8
//   ZATVOR_BURNER2_STATE: AT %MW408
//   OPEN_ZATVOR2: AT %MX404.7
ZATVOR_BURNER2(
    G_EMER := ERR_GAZ OR FIRE,
    ERR_AZ := FALSE,
    AUTO_MODE := ZATVOR2_AUTO,
    HAND_MODE := NOT ZATVOR2_AUTO,
    OPEN_VALVE := BTN_OPEN_ZATVOR2,
    CLOSE_VALVE := BTN_CLOSE_ZATVOR2,
    K_VALVE_OPENED := ZATVOR2_OPENED,
    K_VALVE_CLOSED := ZATVOR2_CLOSED,
    CYCLE_OPEN := ZATVOR_BURNER2_CYCLE_OPEN,
    CYCLE_CLOSE := ZATVOR_BURNER2_CYCLE_CLOSE,
    RESET_ERR := RESET_ERR,
    RUN_TO_CLOSE => CLOSE_ZATVOR2,
    valve_state => ZATVOR_BURNER2_STATE); // VALVE
OPEN_ZATVOR2 := ZATVOR_BURNER2.RUN_TO_OPEN;

// NETWORK 10
//   ZATVOR2_AUTO: AT %MX424.3
//   ZATVOR2_OPENED: AT %MX402.8
//   BTN_CLOSE_ZATVOR2: AT %MX410.7
//   BTN_OPEN_ZATVOR2: AT %MX410.6
_rt3(CLK := BTN_CLOSE_ZATVOR2);
BTN_OPEN_ZATVOR2 R= ZATVOR2_AUTO OR NOT ZATVOR_BURNER2.RR OR ZATVOR2_OPENED OR _rt3.Q;

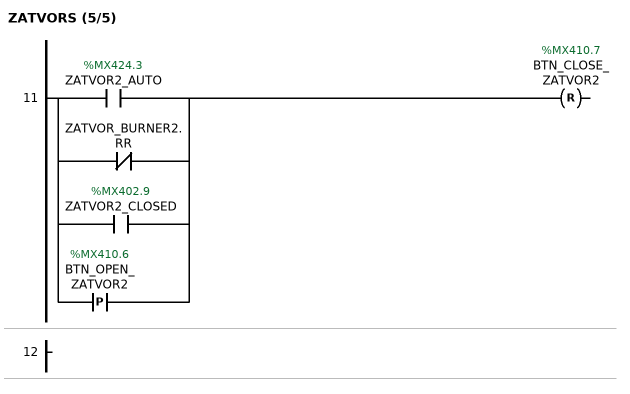
// NETWORK 11
//   ZATVOR2_AUTO: AT %MX424.3
//   ZATVOR2_CLOSED: AT %MX402.9
//   BTN_OPEN_ZATVOR2: AT %MX410.6
//   BTN_CLOSE_ZATVOR2: AT %MX410.7
_rt4(CLK := BTN_OPEN_ZATVOR2);
BTN_CLOSE_ZATVOR2 R= ZATVOR2_AUTO OR NOT ZATVOR_BURNER2.RR OR ZATVOR2_CLOSED OR _rt4.Q;

// NETWORK 12

END_PROGRAM

// MyController/Application/MB_OUT
PROGRAM MB_OUT
VAR

END_VAR

MW128:=POSITION_VALVE_PEREPUSK;
MW129:=POSITION_VALVE_HEATER; 

FREQUENCY_M1:=PCH_PUMP_M1_ZADANIE;
FREQUENCY_M2:=PCH_PUMP_M2_ZADANIE;
FREQUENCY_M7:=PCH_PUMP_M7_ZADANIE;

//FREQUENCY_M1:=FREQ_M1; // %MW134: INT
//FREQUENCY_M2:=FREQ_M2; // %MW135: INT
//FREQUENCY_M7:=FREQ_M7; // %MW136: INT

(*
MW200.0:=ERR_PCH_PUMP_CYRCULATION;
MW200.1:=ERR_PUMP1_CYRCULATION;
MW200.2:=ERR_PUMP2_CYRCULATION;
MW200.3:=ERR_PCH_PUMP1_NET;
MW200.4:=ERR_PCH_PUMP2_NET;
MW200.5:=ERR_M3_FEEDER;
MW200.6:=ERR_M4_FEEDER;
MW200.7:=VALVE_GAZ_OPENED;
MW200.8:=VALVE_GAZ_CLOSED;
MW200.9:=ERR_DEGAZATOR;
MW200.10:=FIRE;
MW200.11:=BREAKE;
MW200.12:=N0_SECURITY;
MW200.13:=SECURITY;
MW200.14:=ERR_GAZ;
MW200.15:=ERR_BURNER1;

MW201.0:=ERR_BURNER2;
MW201.1:=BURNER2_WORKS;
MW201.2:=DYMOHOD1_OPENED;
MW201.3:=DYMOHOD1_CLOSED;
MW201.4:=ZATVOR1_OPENED;
MW201.5:=ZATVOR1_CLOSED;
MW201.6:=DYMOHOD2_OPENED;
MW201.7:=DYMOHOD2_CLOSED;
MW201.8:=ZATVOR2_OPENED;
MW201.9:=ZATVOR2_CLOSED;
MW201.10:=FEEDER_OPENED;
MW201.11:=FEEDER_CLOSED;
MW201.12:=HVO_OPENED;
MW201.13:=HVO_CLOSED;
MW201.14:=PEREPUSK_OPENED;
MW201.15:=PEREPUSK_CLOSED;

MW202.0:=HEATER_CLOSED;
MW202.1:=OPEN_DYMOHOD1;
MW202.2:=CLOSE_DYMOHOD1;
MW202.3:=OPEN_ZATVOR1;
MW202.4:=CLOSE_ZATVOR1;
MW202.5:=OPEN_DYMOHOD2;
MW202.6:=CLOSE_DYMOHOD2;
MW202.7:=OPEN_ZATVOR2;
MW202.8:=CLOSE_ZATVOR2;
MW202.9:=OPEN_FEEDER;
MW202.10:=CLOSE_FEEDER;
MW202.11:=OPEN_HVO;
MW202.12:=CLOSE_HVO;
MW202.13:=OPEN_PEREPUSK;
MW202.14:=CLOSE_PEREPUSK;
MW202.15:=OPEN_HEATER;

MW203.0:=CLOSE_HEATER;
MW203.1:=BURNER1_WORKS;
MW203.2:=HEATER_OPENED;
MW203.3:=RUN_PUMP_CYRCULATION;
MW203.4:=RUN_PUMP_CYRCULATION1;
MW203.5:=RUN_PUMP_CYRCULATION2;
MW203.6:=RUN_PUMP1_NET;
MW203.7:=RUN_PUMP2_NET;
MW203.8:=RUN_M3_FEEDER;
MW203.9:=RUN_M4_FEEDER;
MW203.10:=OPEN_GAZ;
MW203.11:=CLOSE_GAZ;
MW203.12:=RUN_SIGNAL_FIRE;
MW203.13:=RUN_SIGNAL_BREAKE;
MW203.14:=RUN_SMALL_FIRE_BURNER1;
MW203.15:=RUN_LARGE_FIRE_BURNER1;

MW204.0:=RUN_SMALL_FIRE_BURNER2;
MW204.1:=RUN_LARGE_FIRE_BURNER2;



MW205.0:=BTN_OPEN_DYMOHOD1;
MW205.1:=BTN_CLOSE_DYMOHOD1;
MW205.2:=BTN_OPEN_ZATVOR1;
MW205.3:=BTN_CLOSE_ZATVOR1;
MW205.4:=BTN_OPEN_DYMOHOD2;
MW205.5:=BTN_CLOSE_DYMOHOD2;
MW205.6:=BTN_OPEN_ZATVOR2;
MW205.7:=BTN_CLOSE_ZATVOR2;
MW205.8:=BTN_OPEN_FEEDER;
MW205.9:=BTN_CLOSE_FEEDER;
MW205.10:=BTN_OPEN_HVO;
MW205.11:=BTN_CLOSE_HVO;
MW205.12:=BTN_OPEN_PEREPUSK;
MW205.13:=BTN_CLOSE_PEREPUSK;
MW205.14:=BTN_OPEN_HEATER;
MW205.15:=BTN_CLOSE_HEATER;

MW206.0:=BTN_RUN_PUMP_CYRCULATION;
MW206.1:=BTN_RUN_PUMP_CYRCULATION1;
MW206.2:=BTN_RUN_PUMP_CYRCULATION2;
MW206.3:=BTN_RUN_PUMP1_NET;
MW206.4:=BTN_RUN_PUMP2_NET;
MW206.5:=BTN_RUN_M3_FEEDER;
MW206.6:=BTN_RUN_M4_FEEDER;
MW206.7:=BTN_OPEN_GAZ;
MW206.8:=BTN_CLOSE_GAZ;
MW206.9:=BTN_RUN_SIGNAL_FIRE;*)

MW207.0:=DYMOHOD_BURNER1.ERR_K;
MW207.1:=DYMOHOD_BURNER1.ERR_LT;
MW207.2:=DYMOHOD_BURNER2.ERR_K;
MW207.3:=DYMOHOD_BURNER2.ERR_LT;
MW207.4:=ZATVOR_BURNER1.ERR_K;
MW207.5:=ZATVOR_BURNER1.ERR_LT;
MW207.6:=ZATVOR_BURNER2.ERR_K;
MW207.7:=ZATVOR_BURNER2.ERR_LT;
MW207.8:=FEEDER_PB.ERR_K;
MW207.9:=FEEDER_PB.ERR_LT;
MW207.10:=HEATER_BOILER.ERR_K;

MW207.12:=GAZ_GRU.ERR_K;
MW207.13:=GAZ_GRU.ERR_LT;
MW207.14:=HVO_1.ERR_K;
MW207.15:=HVO_1.ERR_LT;

MW208.0:=PEREPUSK.ERR_K;
MW208.1:=ERR_FLOW_IN_NET;
MW208.2:=PUMP_M7.DA;
MW208.3:=PUMP_M5.DA;
MW208.4:=PUMP_M6.DA;
MW208.5:=PUMP_M1.DA;
MW208.6:=PUMP_M2.DA;
MW208.7:=FEEDER_M3.DA;
MW208.8:=FEEDER_M4.DA;
MW208.9:=BURNER_2.ERR_TEMP_HOT;
MW208.10:=ERR_PRES_GAZ;
MW208.11:=BURNER_1.DA;
MW208.12:=ERR_POSITION_PEREPUSK;
MW208.13:=BURNER_1.ERR_TEMP_HOT;
MW208.14:=BURNER_2.DA;
(*
MW209.0:=ERR_SEN_TT1;
MW209.1:=ERR_SEN_TT2;
MW209.2:=ERR_SEN_TT3;
MW209.3:=ERR_SEN_TT4;
MW209.4:=ERR_SEN_TT5;
MW209.5:=ERR_SEN_TT6;
MW209.6:=ERR_SEN_TT7;
MW209.7:=ERR_SEN_TT8;
MW209.8:=ERR_SEN_TT9;
MW209.9:=ERR_SEN_TT10;
MW209.10:=ERR_SEN_TT11;
MW209.11:=ERR_SEN_TT12;
MW209.12:=ERR_SEN_TT13;
MW209.13:=ERR_SEN_TT14;
MW209.14:=ERR_SEN_TT15;
MW209.15:=ERR_SEN_TT16;

MW210.0:=ERR_SEN_PT1;
MW210.1:=ERR_SEN_PT2;
MW210.2:=ERR_SEN_PT3;
MW210.3:=ERR_SEN_PT4;
MW210.4:=ERR_SEN_PT5;
MW210.5:=ERR_SEN_PT6;
MW210.6:=ERR_SEN_PT7;
MW210.7:=ERR_SEN_PT8;
MW210.8:=ERR_SEN_PT9;
MW210.9:=ERR_SEN_PT10;
MW210.10:=ERR_SEN_PT11;
MW210.11:=ERR_SEN_PT01;
MW210.12:=ERR_TRMST_BURNER;
MW210.13:=DA_ALL;*)

END_PROGRAM

// MyController/Application/OUT_PIN
PROGRAM OUT_PIN
VAR

END_VAR

//ВЫХОДЫ МОДУЛЯ А1
Y0:=OPEN_DYMOHOD1;
Y1:=CLOSE_DYMOHOD1;
Y2:=OPEN_ZATVOR1;
Y3:=CLOSE_ZATVOR1;
Y4:=OPEN_DYMOHOD2;
Y5:=CLOSE_DYMOHOD2;
Y6:=OPEN_ZATVOR2;
Y7:=CLOSE_ZATVOR2;
Y8:=OPEN_FEEDER;
Y9:=CLOSE_FEEDER;
Y10:=OPEN_HVO;
Y11:=CLOSE_HVO;
Y12:=OPEN_PEREPUSK;
Y13:=CLOSE_PEREPUSK;
Y14:=OPEN_HEATER;
Y15:=CLOSE_HEATER;

//ВЫХОДЫ МОДУЛЯ А1.3
IY0:=RUN_PUMP_CYRCULATION;
IY1:=RUN_PUMP_CYRCULATION1;
IY2:=RUN_PUMP_CYRCULATION2;
IY3:=RUN_PUMP1_NET;
IY4:=RUN_PUMP2_NET;
IY5:=RUN_M3_FEEDER;
IY6:=RUN_M4_FEEDER;
IY7:=OPEN_GAZ;
IY8:=CLOSE_GAZ;
IY9:=RUN_SIGNAL_FIRE;
IY10:=RUN_SIGNAL_BREAKE;
IY11:=START_STOP_BURNER1;
IY12:=START_STOP_BURNER2;
IY13:=RUN_LARGE_FIRE_BURNER1;
IY14:=RUN_SMALL_FIRE_BURNER1;
IY15:=RUN_LARGE_FIRE_BURNER2;
IY16:=RUN_SMALL_FIRE_BURNER2;
//IY17:=RUN_LIGHT_KOLONNA;
IY18:=RUN_HAND_MODE_PUMPS;
IY19:=RUN_HAND_MODE_BOILERS;
IY20:=RUN_HAND_MODE_VALVES;


IY25:=RUN_LIGHT_KOLONNA;

END_PROGRAM

// MyController/Application/get_data_from_gaz_korr
PROGRAM get_data_from_gaz_korr
VAR
END_VAR

// NETWORK 1

END_PROGRAM

// MyController/Application/A_TESTS/zadanie_for_pch_m7
PROGRAM zadanie_for_pch_m7
VAR
	ZADANIE_FOR_PCH_M5_M6: INT;
END_VAR

(*//УВЕЛИЧЕВАЯ ИЛИ УМЕНЬШАЯ ЧАСТОТУ М7 МЫ ПОДДЕРЖИВАЕМ ЗАДАННУЮ ТЕМПЕРАТУРУ НА ВХОДЕ КОТЛА2
IF TT7_WTR_IN_2<((ZADANIE_TMP_BURNER_2*20)/100)//ТЕМПЕРАТУРА НА ВХОДЕ КОТЛА ДОЛЖНА БЫТЬ НА 20% МЕНЬШЕ ЧЕМ НА ВЫХОДЕ
	THEN IF PCH_PUMP_M7_ZADANIE<50
			THEN 
				IF AUTO_MODE=1
					THEN PCH_PUMP_M7_ZADANIE:=PCH_PUMP_M7_ZADANIE+1;
					ELSE PCH_PUMP_M7_ZADANIE:=MANUAL_ZADANIE_FOR_PCH_M7;
				END_IF
					
		END_IF
	ELSE IF PCH_PUMP_M7_ZADANIE>0
			THEN 
				IF AUTO_MODE=1
					THEN PCH_PUMP_M7_ZADANIE:=PCH_PUMP_M7_ZADANIE-1;
					ELSE PCH_PUMP_M7_ZADANIE:=MANUAL_ZADANIE_FOR_PCH_M7;
				END_IF
		END_IF
END_IF

 *)

END_PROGRAM

// A_TESTS/zadanie_for_pch_m7
PROGRAM zadanie_for_pch_m7
VAR
	ZADANIE_FOR_PCH_M5_M6: INT;
END_VAR

(*//УВЕЛИЧЕВАЯ ИЛИ УМЕНЬШАЯ ЧАСТОТУ М7 МЫ ПОДДЕРЖИВАЕМ ЗАДАННУЮ ТЕМПЕРАТУРУ НА ВХОДЕ КОТЛА2
IF TT7_WTR_IN_2<((ZADANIE_TMP_BURNER_2*20)/100)//ТЕМПЕРАТУРА НА ВХОДЕ КОТЛА ДОЛЖНА БЫТЬ НА 20% МЕНЬШЕ ЧЕМ НА ВЫХОДЕ
	THEN IF PCH_PUMP_M7_ZADANIE<50
			THEN 
				IF AUTO_MODE=1
					THEN PCH_PUMP_M7_ZADANIE:=PCH_PUMP_M7_ZADANIE+1;
					ELSE PCH_PUMP_M7_ZADANIE:=MANUAL_ZADANIE_FOR_PCH_M7;
				END_IF
					
		END_IF
	ELSE IF PCH_PUMP_M7_ZADANIE>0
			THEN 
				IF AUTO_MODE=1
					THEN PCH_PUMP_M7_ZADANIE:=PCH_PUMP_M7_ZADANIE-1;
					ELSE PCH_PUMP_M7_ZADANIE:=MANUAL_ZADANIE_FOR_PCH_M7;
				END_IF
		END_IF
END_IF

 *)

END_PROGRAM

// MyController/Application/A_TESTS/zadanie_m7
PROGRAM zadanie_m7
VAR
	PID_M7: PID;
END_VAR

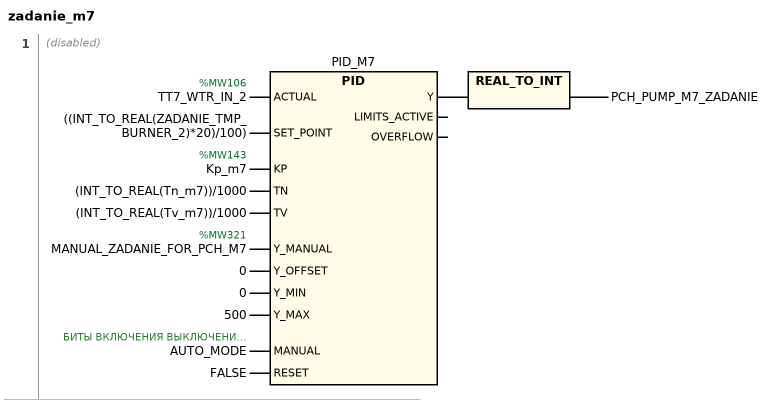
// NETWORK 1 (disabled)
//   TT7_WTR_IN_2: AT %MW106
//   Kp_m7: AT %MW143
//   MANUAL_ZADANIE_FOR_PCH_M7: AT %MW321
//   AUTO_MODE: БИТЫ ВКЛЮЧЕНИЯ ВЫКЛЮЧЕНИЯ МЕХАНИЗМОВ ========== КОНЕЦ ======
// PID_M7(
//     ACTUAL := TT7_WTR_IN_2,
//     SET_POINT := ((INT_TO_REAL(ZADANIE_TMP_BURNER_2)*20)/100),
//     KP := Kp_m7,
//     TN := (INT_TO_REAL(Tn_m7))/1000,
//     TV := (INT_TO_REAL(Tv_m7))/1000,
//     Y_MANUAL := MANUAL_ZADANIE_FOR_PCH_M7,
//     Y_OFFSET := 0,
//     Y_MIN := 0,
//     Y_MAX := 500,
//     MANUAL := AUTO_MODE,
//     RESET := FALSE); // PID
// PCH_PUMP_M7_ZADANIE := REAL_TO_INT(PID_M7.Y);

END_PROGRAM

// A_TESTS/zadanie_m7
PROGRAM zadanie_m7
VAR
	PID_M7: PID;
END_VAR

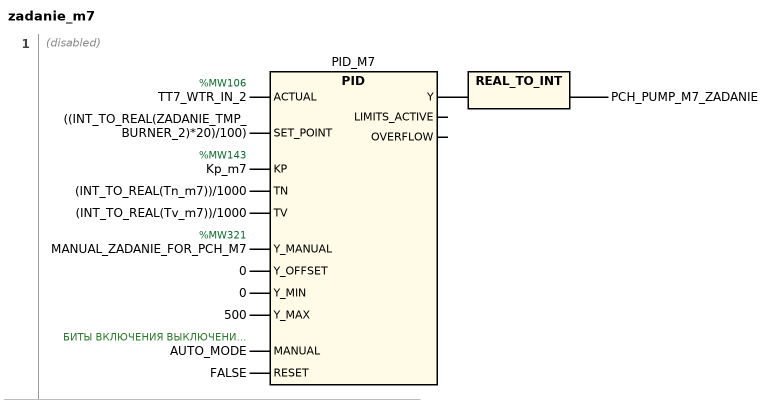
// NETWORK 1 (disabled)
//   TT7_WTR_IN_2: AT %MW106
//   Kp_m7: AT %MW143
//   MANUAL_ZADANIE_FOR_PCH_M7: AT %MW321
//   AUTO_MODE: БИТЫ ВКЛЮЧЕНИЯ ВЫКЛЮЧЕНИЯ МЕХАНИЗМОВ ========== КОНЕЦ ======
// PID_M7(
//     ACTUAL := TT7_WTR_IN_2,
//     SET_POINT := ((INT_TO_REAL(ZADANIE_TMP_BURNER_2)*20)/100),
//     KP := Kp_m7,
//     TN := (INT_TO_REAL(Tn_m7))/1000,
//     TV := (INT_TO_REAL(Tv_m7))/1000,
//     Y_MANUAL := MANUAL_ZADANIE_FOR_PCH_M7,
//     Y_OFFSET := 0,
//     Y_MIN := 0,
//     Y_MAX := 500,
//     MANUAL := AUTO_MODE,
//     RESET := FALSE); // PID
// PCH_PUMP_M7_ZADANIE := REAL_TO_INT(PID_M7.Y);

END_PROGRAM

// MyController/Application/A_TESTS/zadanie_m1_m2
PROGRAM zadanie_m1_m2
VAR
	//PID_M1_M2: PID;
END_VAR
VAR // added by the converter: edge detectors and wires of the graphical bodies
    _w1 : INT;
END_VAR

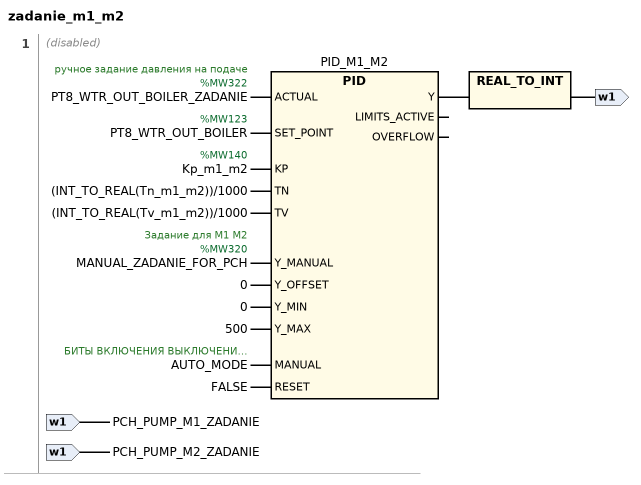
// NETWORK 1 (disabled)
//   PT8_WTR_OUT_BOILER_ZADANIE: ручное задание давления на подаче | AT %MW322
//   PT8_WTR_OUT_BOILER: AT %MW123
//   Kp_m1_m2: AT %MW140
//   MANUAL_ZADANIE_FOR_PCH: Задание для М1 М2 | AT %MW320
//   AUTO_MODE: БИТЫ ВКЛЮЧЕНИЯ ВЫКЛЮЧЕНИЯ МЕХАНИЗМОВ ========== КОНЕЦ ======
// PID_M1_M2(
//     ACTUAL := PT8_WTR_OUT_BOILER_ZADANIE,
//     SET_POINT := PT8_WTR_OUT_BOILER,
//     KP := Kp_m1_m2,
//     TN := (INT_TO_REAL(Tn_m1_m2))/1000,
//     TV := (INT_TO_REAL(Tv_m1_m2))/1000,
//     Y_MANUAL := MANUAL_ZADANIE_FOR_PCH,
//     Y_OFFSET := 0,
//     Y_MIN := 0,
//     Y_MAX := 500,
//     MANUAL := AUTO_MODE,
//     RESET := FALSE); // PID
// _w1 := REAL_TO_INT(PID_M1_M2.Y);
// PCH_PUMP_M1_ZADANIE := _w1;
// PCH_PUMP_M2_ZADANIE := _w1;

END_PROGRAM

// A_TESTS/zadanie_m1_m2
PROGRAM zadanie_m1_m2
VAR
	//PID_M1_M2: PID;
END_VAR
VAR // added by the converter: edge detectors and wires of the graphical bodies
    _w1 : INT;
END_VAR

